// TIA Portal V20 export
DATA_BLOCK "SP506"   // DB234
// stored: MemoryReserve 100
   VAR
      "PHMI EMERGENCY STOP CH.A" : Bool := TRUE;
      "PHMI ENABLE SWITCH CH.A" : Bool := FALSE;
      SPARE : Bool := FALSE;
      SPARE_1 : Bool := FALSE;
      "PHMI EMERGENCY STOP CH.B" : Bool := FALSE;
      "PHMI ENABLE SWITCH CH.B" : Bool := FALSE;
   END_VAR
BEGIN
END_DATA_BLOCK
